Staubli VAL3: SWAP.dtx

public trsf trVision[3]
public trsf trWinCenter
public trsf trWinDown[2]
public trsf trWinMiddle
public trsf trWinUp[2]
public configRx cVision[3]
public configRx cWinCenter
public configRx cWinDown[2]
public configRx cWinMiddle
public configRx cWinUp[2]
public configRs cVisionRS[3]
public configRs cWinCenterRS
public configRs cWinDownRS[2]
public configRs cWinMiddleRS
public configRs cWinUpRS[2]
